// TIA Portal V18 export
FUNCTION_BLOCK "FB_Step"   // FB5002, LAD
{ S7_Optimized_Access := 'TRUE' }
VERSION : 0.1
// stored: AutoNumber false, IsIECCheckEnabled false, IsRetainMemResEnabled false, MemoryReserve 100, SetENOAutomatically false, UDAEnableTagReadback false
   VAR_INPUT
      I_bRun : Bool;   // 运行条件
   END_VAR
   VAR
      sCurrNo : UInt;   // 当前步号
      sNextNo : UInt;   // 下一步号
      sPls : Bool;   // 步序脉冲
      sCondition : Bool;   // 完成条件
      sRunJump : Bool;   // 与输入的运行条件并行
      sTON : TON_TIME;
      sDealyTime { S7_SetPoint := 'True'} : Time;
      sTempNo : UInt;
      bInitialization : Bool;   // 初始化
   END_VAR
   VAR_TEMP   // added for the SCL form of the ladder/FBD networks
      _w1 : Bool;
   END_VAR
BEGIN

REGION Network 1
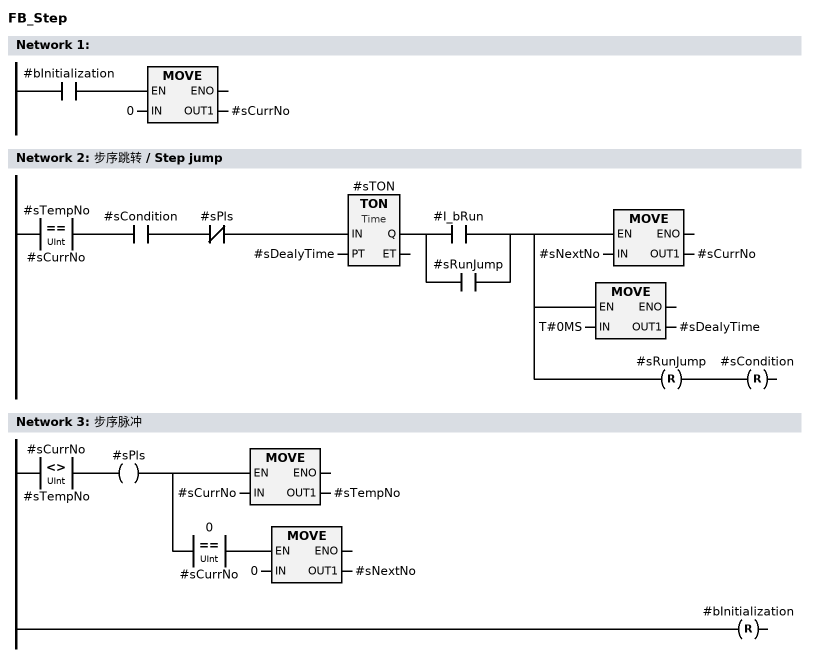
   RUNG wire#powerrail
      Contact( #bInitialization )
      Move(in := 0, out1 => #sCurrNo)
   END_RUNG
   // the same network as SCL:
   IF #bInitialization THEN #sCurrNo := 0; END_IF;
END_REGION

REGION Network 2: 步序跳转 / Step jump
   RUNG wire#powerrail
      { S7_Templates := "SrcType := UInt" } EQ_Contact(in1 := #sTempNo, in2 := #sCurrNo)
      Contact( #sCondition )
      I_Contact( #sPls )
      { S7_Templates := "time_type := Time" } #sTON.TON(pt := #sDealyTime, et =>)
      wire#w1
      Contact( #I_bRun )
      wire#w2
      Move(in := #sNextNo, out1 => #sCurrNo)
   END_RUNG
   RUNG wire#w1
      Contact( #sRunJump )
   END_RUNG wire#w2
   RUNG wire#w2
      Move(in := T#0MS, out1 => #sDealyTime)
   END_RUNG
   RUNG wire#w2
      R_Coil( #sRunJump )
      R_Coil( #sCondition )
   END_RUNG
   // the same network as SCL:
   #sTON(IN := (#sTempNo = #sCurrNo) AND #sCondition AND NOT #sPls, PT := #sDealyTime);   // TON
   IF #sTON.Q AND (#I_bRun OR #sRunJump) THEN
       #sCurrNo := #sNextNo;
       #sDealyTime := T#0MS;
   END_IF;
   #_w1 := #sTON.Q AND (#I_bRun OR #sRunJump);
   IF #_w1 THEN
       #sRunJump := FALSE;
       #sCondition := FALSE;
   END_IF;
END_REGION

REGION Network 3: 步序脉冲
   RUNG wire#powerrail
      { S7_Templates := "SrcType := UInt" } NE_Contact(in1 := #sCurrNo, in2 := #sTempNo)
      Coil( #sPls )
      wire#w1
      Move(in := #sCurrNo, out1 => #sTempNo)
   END_RUNG
   RUNG wire#w1
      { S7_Templates := "SrcType := UInt" } EQ_Contact(in1 := 0, in2 := #sCurrNo)
      Move(in := 0, out1 => #sNextNo)
   END_RUNG
   RUNG wire#powerrail
      R_Coil( #bInitialization )
   END_RUNG
   // the same network as SCL:
   #sPls := #sCurrNo <> #sTempNo;
   IF #sPls THEN #sTempNo := #sCurrNo; END_IF;
   IF #sPls AND (0 = #sCurrNo) THEN #sNextNo := 0; END_IF;
   #bInitialization := FALSE;
END_REGION
END_FUNCTION_BLOCK
